FUNCTION_BLOCK FB_MyNewConfigurationAddTE EXTENDS FB_Base IMPLEMENTS ITF_MCConfiguration
VAR

END_VAR

METHOD AddTopElementToLogger : BOOL
GVL_TopElement1.fbTopElement1.JoinTheLogger ();
GVL_TopElement2.fbTopElement2.JoinTheLogger ();
END_METHOD

(*			
	EVERDE sp. z o.o.
	Rafał Osajda		29.10.2025		TC 4024.66
	Dodawanie TopElementu do systemu
*)
METHOD AddTopElementToMachineControl : BOOL
VAR_INPUT
	itfMachineControl	: ITF_MCMachineControlConfigure;
END_VAR
THIS^.SetText (eLocation := E_BaseLocation.pl, wsDescription := "TopElement 1 pl");
THIS^.SetText (eLocation := E_BaseLocation.en, wsDescription := "TopElement 1 en");
THIS^.SetText (eLocation := E_BaseLocation.de, wsDescription := "TopElement 1 de");
GVL_TopElement1.fbTopElement1.SetName (stName := THIS^.GetTexts ());
itfMachineControl.AddTopElementFromConfiguration (fbTopElement	:= GVL_TopElement1.fbTopElement1);

THIS^.SetText (eLocation := E_BaseLocation.pl, wsDescription := "TopElement 2 pl");
THIS^.SetText (eLocation := E_BaseLocation.en, wsDescription := "TopElement 2 en");
THIS^.SetText (eLocation := E_BaseLocation.de, wsDescription := "TopElement 2 de");
GVL_TopElement1.fbTopElement1.SetName (stName := THIS^.GetTexts ());
itfMachineControl.AddTopElementFromConfiguration (fbTopElement	:= GVL_TopElement2.fbTopElement2);
END_METHOD

METHOD SetStartMode : BOOL
VAR_INPUT
	itfMachineControl	: ITF_MCMachineControlConfigure;
END_VAR
END_METHOD

METHOD StateAndModes : BOOL
VAR_INPUT
	itfMachineControl	: ITF_MCMachineControlConfigure;
END_VAR
END_METHOD

END_FUNCTION_BLOCK

(* stored: Version 1.1.0.1, ProductVersion 3.1.4024.15
   POU FB_MyNewConfigurationAddTE: Id {deb53b3d-9e12-46d3-b5d1-c50be418a5c2}, SpecialFunc None
   Method AddTopElementToLogger: Id {1f68059a-854c-4b77-869d-6d14a3d68622}
   Method AddTopElementToMachineControl: Id {14c2a0df-b97e-48ab-8674-34192113ffc6}
   Method SetStartMode: Id {503f7887-fe7e-43b2-afe8-42df368491ab}
   Method StateAndModes: Id {eaff7a1f-24dd-4234-bac4-3b82e13d6de6} *)
